(* IEC 61131-3 sources: Hydro-Leak-Detection/src/POUs, 4 files *)

(* ---- F_ISO5208LimitMlMin.st ---- *)
(*
    F_ISO5208LimitMlMin

    Allowable liquid leakage rate for a valve, in mL/min, from its nominal bore
    and ISO 5208 rate class.

    ISO 5208 expresses liquid rates as a coefficient per unit of nominal bore
    in mm3/s. Conversion to mL/min:

        1 mm3/s = 0.001 mL/s = 0.06 mL/min

    !! The coefficients in GVL_HydroLeak are PLACEHOLDERS and this function    !!
    !! therefore returns 0.0 for every class until they are populated from the !!
    !! controlled copy of ISO 5208. Returning zero is deliberate: it fails     !!
    !! every valve rather than passing one against an invented limit. Do not   !!
    !! "fix" that by guessing values.                                          !!

    Rate A is handled separately -- it is bounded by the rig noise floor from
    the Stage 4.1 blank test, not by a bore-scaled coefficient.
*)
FUNCTION F_ISO5208LimitMlMin : REAL
VAR_INPUT
    eClass  : E_ISO5208Class;
    rDN_mm  : REAL;
END_VAR
VAR CONSTANT
    c_rMm3PerSec_To_MlPerMin : REAL := 0.06;
END_VAR
VAR
    rCoeff : REAL;
END_VAR

IF rDN_mm <= 0.0 THEN
    F_ISO5208LimitMlMin := 0.0;
    RETURN;
END_IF

CASE eClass OF
    E_ISO5208Class.RATE_A:
        (* Noise-floor bounded, not bore-scaled. *)
        F_ISO5208LimitMlMin := GVL_HydroLeak.c_rRateA_NoiseFloorMlMin;
        RETURN;

    E_ISO5208Class.RATE_B:
        rCoeff := GVL_HydroLeak.c_rISO5208_RateB;

    E_ISO5208Class.RATE_C:
        rCoeff := GVL_HydroLeak.c_rISO5208_RateC;

    E_ISO5208Class.RATE_D:
        rCoeff := GVL_HydroLeak.c_rISO5208_RateD;
ELSE
    rCoeff := 0.0;
END_CASE

F_ISO5208LimitMlMin := rCoeff * rDN_mm * c_rMm3PerSec_To_MlPerMin;

(* ---- F_MinHoldMinutes.st ---- *)
(*
    F_MinHoldMinutes

    Minimum pressurised hold duration for the measurement to be trustworthy
    against a given acceptance threshold.

    Thermal zero drift is a fixed MASS error accumulated over the hold, not a
    rate error. Expressed as a rate it therefore divides by the hold duration:

        rate error (mg/min) = total drift (mg) / hold (min)

    So the hold needed to keep drift below an acceptable fraction of the
    threshold is:

        T_min = k * TotalDrift_mg / (Threshold_mL_min * density_g_mL)

    where k = 1 / acceptable_fraction  (k = 5 for a 20 % error allowance).

    This is why "hold duration varies by valve size and spec" cannot simply be
    accepted as an input. The acceptance threshold scales with nominal bore, so
    a small-bore valve on a tight rate class needs a LONGER hold than a large
    one -- the opposite of what test schedules usually assume. Rather than
    trusting the schedule, the program computes what this rig actually needs
    and refuses to issue a verdict on a hold that was too short.

    TotalDrift_mg comes from the Stage 4.5 thermal characterisation, not from
    the datasheet: it is the measured mg/degC of the assembled chain multiplied
    by the temperature excursion the vessel actually sees during a hold.

    Worked example -- 1 kg cell, open workshop:
        50 mg/degC * 2 degC = 100 mg total drift
        threshold 0.01 mL/min, k = 5
        T_min = 5 * 100 / (0.01 * 1000 * 0.998) = 50 minutes
*)
FUNCTION F_MinHoldMinutes : REAL
VAR_INPUT
    rThresholdMlMin  : REAL;   (* active ISO 5208 limit for this valve *)
    rTotalDriftMg    : REAL;   (* from Stage 4.5, for the expected excursion *)
    rDensityGPerMl   : REAL;
    rErrorAllowance  : REAL;   (* e.g. 0.20 for 20 % *)
END_VAR
VAR
    rK : REAL;
END_VAR

(* A zero or negative threshold means Rate A bounded by the noise floor, or an
   unpopulated ISO 5208 coefficient. Neither can produce a meaningful hold
   requirement, so demand the configured maximum rather than returning zero --
   returning zero would silently declare any hold long enough. *)
IF rThresholdMlMin <= 0.0 OR rDensityGPerMl <= 0.0 OR rErrorAllowance <= 0.0 THEN
    F_MinHoldMinutes := GVL_HydroLeak.c_rMaxPracticalHoldMin;
    RETURN;
END_IF

rK := 1.0 / rErrorAllowance;

F_MinHoldMinutes := (rK * rTotalDriftMg)
                    / (rThresholdMlMin * rDensityGPerMl * 1000.0);

(* ---- FB_LeastSquaresSlope.st ---- *)
(*
    FB_LeastSquaresSlope

    Rolling-window least-squares fit of mass against time. Reusable -- nothing
    in here is leak-specific.

    Why a slope and not a difference of consecutive samples:
    differencing amplifies noise (the difference of two noisy samples has ~1.4x
    the noise of one) and carries no averaging. A regression over N samples
    suppresses zero-mean noise by ~sqrt(N) and, more importantly, is blind to
    every CONSTANT offset in the chain -- cell zero balance, tare error, vessel
    mass, absolute calibration error. Only drift occurring inside the window
    survives into the result.

    Accumulators are LREAL. Sum-of-squares terms grow as n*t^2; over a
    60-minute window at 1 Hz that exceeds the ~7 significant digits a 32-bit
    REAL carries, and the fit silently degrades rather than failing.

    The window is maintained incrementally (add new, subtract outgoing) for
    O(1) cost per cycle. Repeated subtraction accumulates rounding error over
    long runs, so the sums are fully recomputed from the buffer every
    c_udiRebaseInterval updates.

    rR2 is reported so the caller can reject a window that is not usefully
    linear. Unsettled creep, a knocked rig, and float stick-slip all show up as
    a poor fit rather than as an obviously wrong number.
*)
FUNCTION_BLOCK FB_LeastSquaresSlope
VAR_INPUT
    bEnable      : BOOL;
    bReset       : BOOL;
    rTimeSec     : REAL;
    rValue       : REAL;
    uiWindowSize : UINT := 600;
END_VAR
VAR_OUTPUT
    rSlopePerSec : REAL;
    rSlopePerMin : REAL;
    rR2          : REAL;
    rIntercept   : REAL;
    uiCount      : UINT;    (* samples currently in the window *)
    bWindowFull  : BOOL;
    bValid       : BOOL;
END_VAR
VAR CONSTANT
    c_uiMaxWindow        : UINT  := 3600;   (* 1 hour at 1 Hz *)
    c_udiRebaseInterval  : UDINT := 10000;
END_VAR
VAR
    arT      : ARRAY[0..3599] OF LREAL;
    arV      : ARRAY[0..3599] OF LREAL;
    uiHead   : UINT;
    uiN      : UINT;
    uiWin    : UINT;
    udiSince : UDINT;

    lrN, lrSt, lrSv, lrStt, lrSvv, lrStv : LREAL;
    lrSxx, lrSyy, lrSxy, lrSlope : LREAL;
    lrOutT, lrOutV : LREAL;
    i : UINT;
END_VAR

IF bReset THEN
    uiHead := 0;  uiN := 0;  udiSince := 0;
    lrN := 0.0; lrSt := 0.0; lrSv := 0.0;
    lrStt := 0.0; lrSvv := 0.0; lrStv := 0.0;
    rSlopePerSec := 0.0;  rSlopePerMin := 0.0;
    rR2 := 0.0;  rIntercept := 0.0;
    uiCount := 0;  bWindowFull := FALSE;  bValid := FALSE;
    RETURN;
END_IF

(* Clamp the requested window to the allocated buffer. *)
uiWin := uiWindowSize;
IF uiWin > c_uiMaxWindow THEN
    uiWin := c_uiMaxWindow;
END_IF
IF uiWin < 2 THEN
    uiWin := 2;
END_IF

IF bEnable THEN
    (* Evict the oldest sample once the window is full. *)
    IF uiN >= uiWin THEN
        lrOutT := arT[uiHead];
        lrOutV := arV[uiHead];
        lrN    := lrN   - 1.0;
        lrSt   := lrSt  - lrOutT;
        lrSv   := lrSv  - lrOutV;
        lrStt  := lrStt - lrOutT * lrOutT;
        lrSvv  := lrSvv - lrOutV * lrOutV;
        lrStv  := lrStv - lrOutT * lrOutV;
        uiN    := uiN - 1;
    END_IF

    arT[uiHead] := TO_LREAL(rTimeSec);
    arV[uiHead] := TO_LREAL(rValue);
    lrN   := lrN   + 1.0;
    lrSt  := lrSt  + arT[uiHead];
    lrSv  := lrSv  + arV[uiHead];
    lrStt := lrStt + arT[uiHead] * arT[uiHead];
    lrSvv := lrSvv + arV[uiHead] * arV[uiHead];
    lrStv := lrStv + arT[uiHead] * arV[uiHead];

    uiHead := (uiHead + 1) MOD uiWin;
    uiN    := uiN + 1;

    (* Periodic exact rebase against accumulated subtraction error. *)
    udiSince := udiSince + 1;
    IF udiSince >= c_udiRebaseInterval THEN
        udiSince := 0;
        lrN := 0.0; lrSt := 0.0; lrSv := 0.0;
        lrStt := 0.0; lrSvv := 0.0; lrStv := 0.0;
        FOR i := 0 TO uiN - 1 DO
            lrN   := lrN   + 1.0;
            lrSt  := lrSt  + arT[i];
            lrSv  := lrSv  + arV[i];
            lrStt := lrStt + arT[i] * arT[i];
            lrSvv := lrSvv + arV[i] * arV[i];
            lrStv := lrStv + arT[i] * arV[i];
        END_FOR
    END_IF
END_IF

uiCount     := uiN;
bWindowFull := (uiN >= uiWin);

IF lrN < 2.0 THEN
    bValid := FALSE;
    RETURN;
END_IF

lrSxx := lrStt - (lrSt * lrSt) / lrN;
lrSyy := lrSvv - (lrSv * lrSv) / lrN;
lrSxy := lrStv - (lrSt * lrSv) / lrN;

(* Sxx is zero only if every sample in the window shares one timestamp. *)
IF lrSxx <= 0.0 THEN
    bValid := FALSE;
    RETURN;
END_IF

lrSlope      := lrSxy / lrSxx;
rSlopePerSec := LREAL_TO_REAL(lrSlope);
rSlopePerMin := LREAL_TO_REAL(lrSlope * 60.0);
rIntercept   := LREAL_TO_REAL((lrSv - lrSlope * lrSt) / lrN);

(* Syy = 0 is a perfectly flat trace -- a tight valve, not an error. *)
IF lrSyy > 0.0 THEN
    rR2 := LREAL_TO_REAL((lrSxy * lrSxy) / (lrSxx * lrSyy));
ELSE
    rR2 := 1.0;
END_IF

bValid := TRUE;

(* ---- PRG_HydroLeakDetection.st ---- *)
(*
    PRG_HydroLeakDetection

    Gravimetric micro-leak detection for hydrostatic valve testing.
    Target sensitivity 0.01 mL/min == 10 mg/min of captured water.

    Replaces PR2_Leak_Detection, which is retired rather than extended. Its
    tare and settle pattern carried over; its scaling and its output did not.

    Changes from PR2, and why each one matters:

    1. Raw input DINT via GVL_IO, not INT. Reading the 24-bit ELM3148 as 16
       bits gave 30.5 mg/count -- a full 20-minute signal spanning six counts.

    2. Scaling endpoints from the Stage 2.4 bench calibration, not 0/32767.
       32767 is a 16-bit convention, not a property of this converter.

    3. Output is a RATE, fitted by least squares over a rolling window. PR2
       reported an instantaneous mass difference and labelled it leak volume.
       Acceptance criteria are written as rates, and a slope cancels every
       constant offset in the chain.

    4. Threshold computed per test from valve DN and ISO 5208 rate class.

    5. Settle time minutes, not 3 s, with tare at the END of it. Three seconds
       damps suspension swing; creep decays over minutes and mimics a leak.

    6. No negative clamp. PR2 clamped at zero, which rectifies noise into a
       positive bias -- an apparent leak on a tight valve -- and conceals net
       mass LOSS, the signature of an unsealed catch vessel. Evaporation from
       an open vessel is 40-85 % of the signal and removes mass, so it biases
       towards PASSING a leaking valve. See docs/measurement-budget.md 2.1.

    7. Fit quality gates the verdict. A disturbed run is a retest, not a pass.

    Corroborating channel B is read and logged but does not yet gate the
    verdict -- that cross-check is defined in docs/commissioning.md Stage 5.3
    and should not be armed until the bench tests establish its noise floor.
*)
PROGRAM PRG_HydroLeakDetection
VAR
    (* --- Per-test inputs, supplied with the valve ID from the HMI --- *)
    bStartTestCycle        : BOOL;
    bOperatorAbort         : BOOL;
    sValveId               : STRING(32);
    rValveDN_mm            : REAL;                     (* nominal bore *)
    eRateClass             : E_ISO5208Class;           (* A / B / C / D *)
    rFluidDensityGPerMl    : REAL := 0.998;
    tHoldDuration          : TIME := T#20M;

    (* --- Scaled process values --- *)
    rAbsoluteMassG         : REAL;
    rTareMassG             : REAL;
    rCapturedMassG         : REAL;    (* may legitimately go negative *)
    rCorroborationEng      : REAL;
    rVesselTempC           : REAL;

    (* --- Result --- *)
    rLeakRateMlMin         : REAL;
    rActiveThresholdMlMin  : REAL;
    rFitR2                 : REAL;
    bResultTrustworthy     : BOOL;
    bLeakWithinLimit       : BOOL;
    bTestComplete          : BOOL;

    (* --- State --- *)
    eState                 : E_LeakState := E_LeakState.IDLE;
    rElapsedSec            : REAL;

    (* --- Instances --- *)
    fbSettleTimer          : TON;
    fbDiscardTimer         : TON;
    fbHoldTimer            : TON;
    fbAlarmDebounce        : TON;
    fbSlope                : FB_LeastSquaresSlope;

    (* --- Scratch --- *)
    rSpanCounts            : REAL;
    bLoopFault             : BOOL;
END_VAR

// =============================================================================
// 1. Loop health
// =============================================================================
(* Under-range means the 4-20 mA loop is open: a pulled cable, a dead
   conditioner, or an XLR backed out of its shell. This must abort the test.
   A broken loop reading 0 mA scales to a large NEGATIVE mass, which a naive
   implementation would report as a very tight valve. *)
bLoopFault := GVL_IO.bChAError OR GVL_IO.bChAUnderrange OR GVL_IO.bChAOverrange;

// =============================================================================
// 2. Scaling -- from the Stage 2.4 two-point calibration
// =============================================================================
rSpanCounts := DINT_TO_REAL(GVL_HydroLeak.c_diChA_Raw_20mA - GVL_HydroLeak.c_diChA_Raw_4mA);

IF rSpanCounts <> 0.0 THEN
    rAbsoluteMassG := (DINT_TO_REAL(GVL_IO.diRawMassChA - GVL_HydroLeak.c_diChA_Raw_4mA)
                       / rSpanCounts) * GVL_HydroLeak.c_rChA_SpanGrams;
ELSE
    rAbsoluteMassG := 0.0;
END_IF

rSpanCounts := DINT_TO_REAL(GVL_HydroLeak.c_diChB_Raw_20mA - GVL_HydroLeak.c_diChB_Raw_4mA);
IF rSpanCounts <> 0.0 THEN
    rCorroborationEng := (DINT_TO_REAL(GVL_IO.diRawCorrobChB - GVL_HydroLeak.c_diChB_Raw_4mA)
                          / rSpanCounts) * GVL_HydroLeak.c_rChB_SpanEng;
ELSE
    rCorroborationEng := 0.0;
END_IF

// =============================================================================
// 3. Acceptance threshold -- per test, from DN and rate class
// =============================================================================
(* ISO 5208 liquid rates are expressed per unit of nominal bore, so the limit
   is recomputed for every valve rather than compiled in. Coefficients live in
   GVL_HydroLeak and are PLACEHOLDERS until verified against the controlled
   copy of the standard -- see that file's header. *)
rActiveThresholdMlMin := F_ISO5208LimitMlMin(eClass := eRateClass, rDN_mm := rValveDN_mm);

// =============================================================================
// 4. Timers -- serviced before the state logic so .Q and .ET are current
// =============================================================================
fbSettleTimer( IN := (eState = E_LeakState.SETTLING), PT := GVL_HydroLeak.c_tSettleTime);
fbDiscardTimer(IN := (eState = E_LeakState.TARED),    PT := GVL_HydroLeak.c_tDiscardAtStart);
fbHoldTimer(   IN := (eState = E_LeakState.TESTING),  PT := tHoldDuration);

// =============================================================================
// 5. Sequence
// =============================================================================
CASE eState OF

    E_LeakState.IDLE:
        bTestComplete      := FALSE;
        bLeakWithinLimit   := FALSE;
        bResultTrustworthy := FALSE;
        rTareMassG         := 0.0;
        rCapturedMassG     := 0.0;
        rLeakRateMlMin     := 0.0;
        rElapsedSec        := 0.0;
        fbSlope(bReset := TRUE);

        IF bStartTestCycle AND NOT bLoopFault THEN
            eState := E_LeakState.SETTLING;
        END_IF

    E_LeakState.SETTLING:
        (* Unpressurised, vessel resting on the cell. Creep decaying. *)
        IF fbSettleTimer.Q THEN
            eState := E_LeakState.TARED;
        END_IF

    E_LeakState.TARED:
        (* Zero captured once, at the end of settling. Then the opening
           minutes of the pressurised hold are discarded so residual creep and
           the thermal transient from pressurisation stay out of the fit. *)
        IF fbDiscardTimer.ET = T#0S THEN
            rTareMassG := rAbsoluteMassG;
        END_IF

        IF fbDiscardTimer.Q THEN
            fbSlope(bReset := TRUE);
            rElapsedSec := 0.0;
            eState      := E_LeakState.TESTING;
        END_IF

    E_LeakState.TESTING:
        (* Elapsed time taken from the timer rather than accumulated by adding
           a nominal cycle time, which drifts against real time. *)
        rElapsedSec := TIME_TO_REAL(fbHoldTimer.ET) / 1000.0;

        IF fbAlarmDebounce.Q THEN
            eState := E_LeakState.ALARM;
        ELSIF fbHoldTimer.Q THEN
            bTestComplete := TRUE;
        END_IF

    E_LeakState.ALARM:
        bTestComplete := TRUE;

    E_LeakState.ABORTED:
        bTestComplete := FALSE;

END_CASE

// =============================================================================
// 6. Captured mass and rate
// =============================================================================
(* Deliberately unclamped. Negative captured mass is real information: the
   vessel is losing water faster than the valve leaks into it, which indicates
   an unsealed vessel or a thermal problem -- not a tight valve. *)
IF eState = E_LeakState.TARED OR eState = E_LeakState.TESTING
   OR eState = E_LeakState.ALARM THEN
    rCapturedMassG := rAbsoluteMassG - rTareMassG;
ELSE
    rCapturedMassG := 0.0;
END_IF

fbSlope(
    bEnable      := (eState = E_LeakState.TESTING),
    bReset       := FALSE,
    rTimeSec     := rElapsedSec,
    rValue       := rCapturedMassG,
    uiWindowSize := GVL_HydroLeak.c_uiSlopeWindowSize
);

rFitR2 := fbSlope.rR2;

IF rFluidDensityGPerMl > 0.0 THEN
    rLeakRateMlMin := fbSlope.rSlopePerMin / rFluidDensityGPerMl;
ELSE
    rLeakRateMlMin := 0.0;
END_IF

// =============================================================================
// 7. Alarm debounce
// =============================================================================
(* The rate must stay over the limit continuously before the state latches.
   A single noisy window must not fail a valve. The window must also be full --
   a slope fitted over three samples is meaningless. *)
fbAlarmDebounce(
    IN := (eState = E_LeakState.TESTING)
          AND fbSlope.bValid
          AND fbSlope.bWindowFull
          AND (rLeakRateMlMin > rActiveThresholdMlMin),
    PT := GVL_HydroLeak.c_tAlarmDebounce
);

// =============================================================================
// 8. Verdict
// =============================================================================
bResultTrustworthy := bTestComplete
                      AND fbSlope.bValid
                      AND fbSlope.bWindowFull
                      AND (rFitR2 >= GVL_HydroLeak.c_rMinR2)
                      AND NOT bLoopFault;

bLeakWithinLimit   := bResultTrustworthy
                      AND (eState <> E_LeakState.ALARM)
                      AND (rLeakRateMlMin <= rActiveThresholdMlMin);

// =============================================================================
// 9. Abort
// =============================================================================
IF bOperatorAbort OR bLoopFault THEN
    IF eState <> E_LeakState.IDLE THEN
        eState := E_LeakState.ABORTED;
    END_IF
END_IF

IF NOT bStartTestCycle THEN
    eState := E_LeakState.IDLE;
END_IF
